FUNCTION_BLOCK sifb_teste
  (* Standard: 61499-2 *)
  (* Version 03-07-12, GASR *)
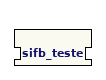
END_FUNCTION_BLOCK
